# EPICS autosave request: gardasoftLED/PP420ProfileChannel_settings.req
$(P):PR$(PROFILE):CH$(CHANNEL):BRIGHTNESS
$(P):PR$(PROFILE):CH$(CHANNEL):DELAY
$(P):PR$(PROFILE):CH$(CHANNEL):TRIG_EDGE
$(P):PR$(PROFILE):CH$(CHANNEL):WIDTH
